(* CODESYS project FB1_AddSub.project

Project tree, tasks and I/O mapping:
  Device : CODESYS Control Win V3, 3S - Smart Software Solutions GmbH, version 3.5.15.30
    application Application
      libraries: Standard, * (System)
      task MainTask (cyclic, interval t#20ms, priority 1) calls PLC_PRG
      task VISU_TASK (cyclic, interval 100 ms, priority 31) calls VisuElems.Visu_Prg
      program PLC_PRG [FBD]
      visualisation Visualization
      function block MyPOU [ST]
  text list GlobalTextList
*)

// Device/Application/PLC_PRG
PROGRAM PLC_PRG
VAR
	MyPOU_0: MyPOU;
	MyPOU_0_Num1: REAL;
	MyPOU_0_Num2: REAL;
	MyPOU_0_AddResult: REAL;
	MyPOU_0_SubResult: REAL;
END_VAR

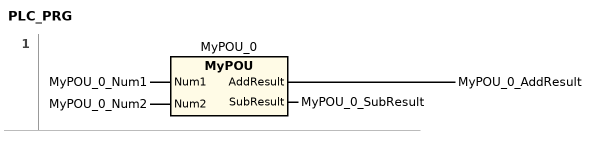
// NETWORK 1
MyPOU_0(Num1 := MyPOU_0_Num1, Num2 := MyPOU_0_Num2, SubResult => MyPOU_0_SubResult); // MyPOU
MyPOU_0_AddResult := MyPOU_0.AddResult;

END_PROGRAM

// Device/Application/MyPOU
FUNCTION_BLOCK MyPOU
VAR_INPUT
	Num1: REAL;
	Num2: REAL;
END_VAR
VAR_OUTPUT
	AddResult : REAL;
	SubResult : REAL;
END_VAR
VAR
END_VAR

AddResult := Num1 + Num2;
SubResult := Num1 - Num2;

END_FUNCTION_BLOCK

// Device/Application/Visualization
VISUALIZATION Visualization  // 2x2
END_VISUALIZATION
